Xinje XDPPro project, PLC1: XD3-24 (software 3.7.17c 2024-04-02)

PROGRAM Ladder

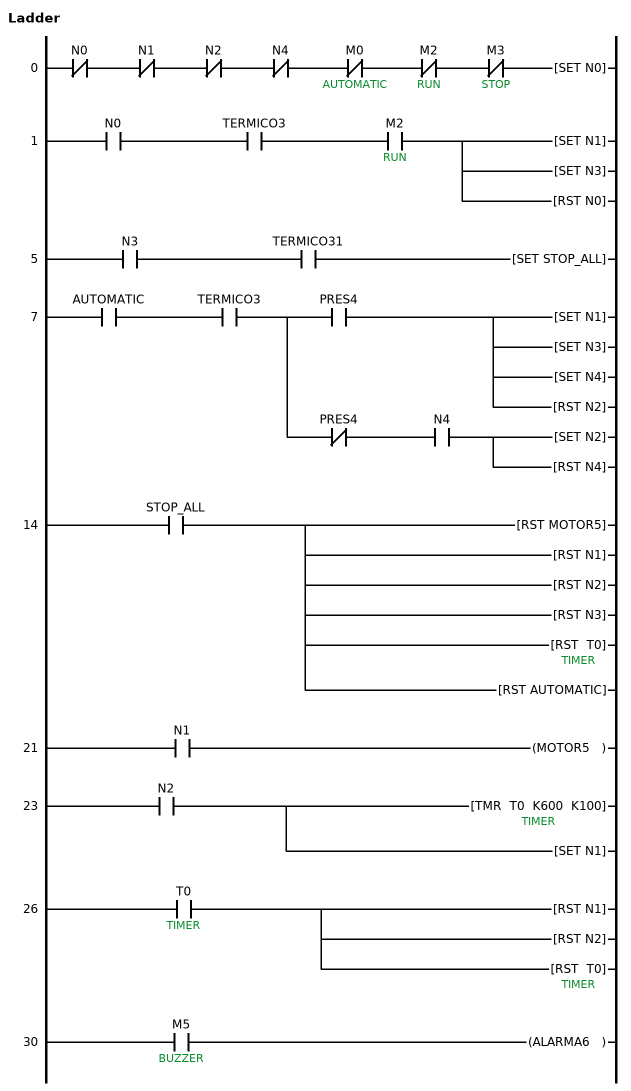
LDI    N0
ANI    N1
ANI    N2
ANI    N4
ANI    M0	; AUTOMATIC
ANI    M2	; RUN
ANI    M3	; STOP
SET    N0
LD     N0
AND    TERMICO3
AND    M2	; RUN
SET    N1
SET    N3
RST    N0
LD     N3
AND    TERMICO31
SET    STOP_ALL
LD     AUTOMATIC
AND    TERMICO3
MPS
AND    PRES4
SET    N1
SET    N3
SET    N4
RST    N2
MPP
ANI    PRES4
AND    N4
SET    N2
RST    N4
LD     STOP_ALL
RST    MOTOR5
RST    N1
RST    N2
RST    N3
RST    T0	; TIMER
RST    AUTOMATIC
LD     N1
OUT    MOTOR5
LD     N2
TMR    T0 K600 K100	; TIMER
SET    N1
LD     T0	; TIMER
RST    N1
RST    N2
RST    T0	; TIMER
LD     M5	; BUZZER
OUT    ALARMA6

COMMENTS (devices not used above)
Y0	MOTOR 5
Y1	ALARMA 6
X0	TERMICO 3 INDICADOR
X1	PRESOSTATO 4
X2	TERMICO 31 SEÑAL
D0	PRESION
ID0	VAC/AMP
TD0	CONTADOR

GLOBAL VARIABLES Global Variable Table
TERMICO3 : BIT	VarType=BIT, VarMap=X0, VarComment=IN
PRES4 : BIT	VarType=BIT, VarMap=X1, VarComment=IN
TERMICO31 : BIT	VarType=BIT, VarMap=X2, VarComment=IN
MOTOR5 : BIT	VarType=BIT, VarMap=Y0, VarComment=OUT
ALARMA6 : BIT	VarType=BIT, VarMap=Y1, VarComment=OUT
AUTOMATIC : BIT	NetworkPublicity=true, VarType=BIT, VarMap=M0, VarComment=M0
RUN : BIT	VarType=BIT, VarMap=M2, VarComment=M2
STOP_ALL : BIT	VarType=BIT, VarMap=M3, VarComment=M3
N0 : BIT	VarType=BIT, VarMap=M6, VarComment=MARCA0
N1 : BIT	VarType=BIT, VarMap=M7, VarComment=MARCA1
N2 : BIT	VarType=BIT, VarMap=M8, VarComment=MARCA2
N3 : BIT	VarType=BIT, VarMap=M9, VarComment=MARCA3
N4 : BIT	VarType=BIT, VarMap=M1, VarComment=CONDICION